FUNCTION_BLOCK E_SEL_UINT (* Event-driven UINT selection *)
  (* Standard: 61499-1; Function: Math; Type: Selection; Description: UINT selection *)
  (* Version 0.0, 2004-09-23, JHC, Rockwell Automation *)
  (* Compiler header: package fb.rt.math; *)
  (* Compiler Java Sun JDK 1.4.2 *)
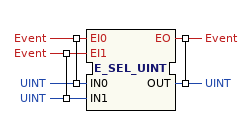
  EVENT_INPUT
    EI0 WITH IN0; (* Select INO *)
    EI1 WITH IN1; (* Select IN1 *)
  END_EVENT
  EVENT_OUTPUT
    EO WITH OUT; (* New selection event *)
  END_EVENT
  VAR_INPUT
    IN0 : UINT; (* Selected by EI0 *)
    IN1 : UINT; (* Selected by EI1 *)
  END_VAR
  VAR_OUTPUT
    OUT : UINT; (* Selected value *)
  END_VAR
END_FUNCTION_BLOCK
